// TIA Portal V20 export
VAR_GLOBAL   // PLC tag table "LKinCtrl_HMI_Editor_Interlocks"
END_VAR
VAR_GLOBAL CONSTANT   // user constants
   LKINCTRL_INTERLOCKID_MOVEPATH_RUNNING : Int := 7001;
END_VAR
